TYPE (* IEC61131-3, Table 14#5 *)
  (* Standard: 1131-3 *)
  (* Version 0.0, 1/8/2024, Cheyan, Schneider Electric, Template *)
  PACKAGE Main;
  {SET_ATTRIBUTE(nxtDataType, KGq6wfCiXsBeHlxye7CIu608a+nl0pPORI0dtNztoWRCF3/wLcc/3fUcieogfuL5MoZOCexFZKjLlqDRxpnKKa/P2zGHmA99mbE0H1MxjlYb9Gog09kpguoYBM5y7X//PNaJMBYTnESNqlHlZuKJzMWQ12cACnhJoVfCmRMo4DhpT+lALlHIn2Y42hllnSHlO+Cvie4vyUd3ROGtjsMnq/3IL42w1oq++pyC2odAP2w=)}
  Quality : STRUCT
    validity : validity;
    detailQual : detailQual;
    source : source;
    test : BOOL;
    operatorBlocked : BOOL;
  END_STRUCT;
END_TYPE
